{attribute 'GeneratedUsingTerminal: EP3744-0041-0016'}
{attribute addProperty BoxType "EP3744-0041-0016"}
{attribute addProperty Id "Set_safe_stateAT %Q*BOOL1"}
{attribute addProperty CRC "1509937735"}
{attribute addProperty Size "1"}
TYPE DEV_Outputs_Device_59FFD247 :
STRUCT
	{attribute addProperty Name "Set_safe_state"}
	Set_safe_state AT %Q* : BOOL;
END_STRUCT
END_TYPE

(* stored: Version 1.2.0.0, ProductVersion 3.1.4024.9
   DUT DEV_Outputs_Device_59FFD247: Id {48f4a858-e66d-4298-ae90-5ad584cb1de0} *)
